PROGRAM Events
VAR
	Send_Start_Event : Send_Event_FB;
	Start_Event  : TcEventEntry := TC_Events.Pelletizer_Events.Start_Button_Event;
	
	Send_Stop_Event : Send_Event_FB;
	Stop_Event  : TcEventEntry := TC_Events.Pelletizer_Events.Stop_Button_Event;
//////////////////////////////////////////////////////////////////////////////////////////////////////////////////
	Send_EmergencyStop_Event : Send_Event_FB;
	EmergencyStop_Event : TcEventEntry := TC_Events.Pelletizer_Events.Emergency_Stop_Set_Event;

	Send_EmergencyStop_Reset_Event : Send_Event_FB;
	EmergencyStop_Reset_Event : TcEventEntry := TC_Events.Pelletizer_Events.Emergency_Stop_Reset_Event;
//////////////////////////////////////////////////////////////////////////////////////////////////////////////////
	Send_Discharge_Chute_NotPresent_Event : Send_Event_FB;
	Discharge_Chute_NotPresent_Event : TcEventEntry := TC_Events.Pelletizer_Events.Discharge_Chute_NotPresent_Event;
	
	Send_Discharge_Chute_Present_Event : Send_Event_FB;
	Discharge_Chute_Present_Event : TcEventEntry := TC_Events.Pelletizer_Events.Discharge_Chute_Present_Event;
//////////////////////////////////////////////////////////////////////////////////////////////////////////////////	
	Send_FeedThroat_NotPresent_Event : Send_Event_FB;
	FeedThroat_NotPresent_Event : TcEventEntry := TC_Events.Pelletizer_Events.FeedThroat_NotPresent_Event;
	
	Send_FeedThroat_Present_Event : Send_Event_FB;
	FeedThroat_Present_Event : TcEventEntry := TC_Events.Pelletizer_Events.FeedThroat_Present_Event;
//////////////////////////////////////////////////////////////////////////////////////////////////////////////////	
	Send_Feedroll_Drive_Fault_Event : Send_Event_FB;
	Feedroll_Drive_Fault_Event : TcEventEntry := TC_Events.Pelletizer_Events.Feedroll_Drive_Fault_Event;
	
	Send_Feedroll_Drive_Fault_Reset_Event : Send_Event_FB;
	Feedroll_Drive_Fault_Reset_Event : TcEventEntry := TC_Events.Pelletizer_Events.Feedroll_Drive_Fault_Reset_Event;
//////////////////////////////////////////////////////////////////////////////////////////////////////////////////	
	Send_Rotor_Drive_Fault_Event : Send_Event_FB;
	Rotor_Drive_Fault_Event : TcEventEntry := TC_Events.Pelletizer_Events.Rotor_Drive_Fault_Event;
	
	Send_Rotor_Drive_Fault_Reset_Event : Send_Event_FB;
	Rotor_Drive_Fault_Reset_Event : TcEventEntry := TC_Events.Pelletizer_Events.Rotor_Drive_Fault_Reset_Event;
//////////////////////////////////////////////////////////////////////////////////////////////////////////////////
	Send_Machine_Shutdown_Event : Send_Event_FB;
	Machine_Shutdown_Event : TcEventEntry := TC_Events.Pelletizer_Events.Machine_Shutdown_Event;	
	
	Send_Machine_PowerOn_Event : Send_Event_FB;
	Machine_PowerOn_Event : TcEventEntry := TC_Events.Pelletizer_Events.Machine_PowerOn_Event;
	First_Scan : BOOL := False;	
END_VAR

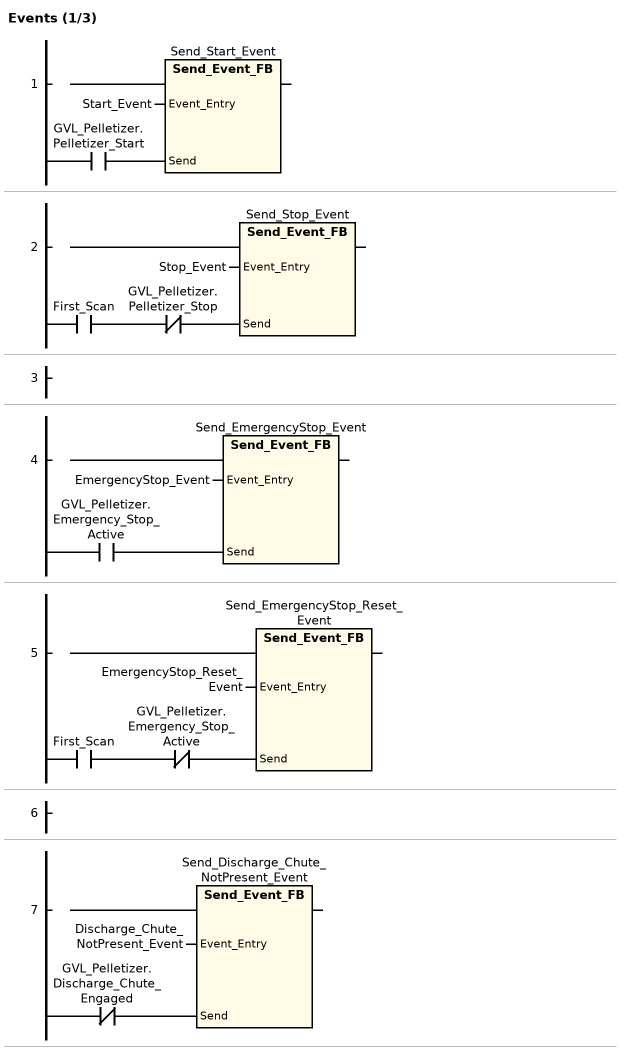
// NETWORK 1
Send_Start_Event(Event_Entry := Start_Event, Send := GVL_Pelletizer.Pelletizer_Start); // Send_Event_FB

// NETWORK 2
Send_Stop_Event(Event_Entry := Stop_Event, Send := First_Scan AND NOT GVL_Pelletizer.Pelletizer_Stop); // Send_Event_FB

// NETWORK 3

// NETWORK 4
Send_EmergencyStop_Event(Event_Entry := EmergencyStop_Event, Send := GVL_Pelletizer.Emergency_Stop_Active); // Send_Event_FB

// NETWORK 5
Send_EmergencyStop_Reset_Event(Event_Entry := EmergencyStop_Reset_Event, Send := First_Scan AND NOT GVL_Pelletizer.Emergency_Stop_Active); // Send_Event_FB

// NETWORK 6

// NETWORK 7
Send_Discharge_Chute_NotPresent_Event(Event_Entry := Discharge_Chute_NotPresent_Event, Send := NOT GVL_Pelletizer.Discharge_Chute_Engaged); // Send_Event_FB

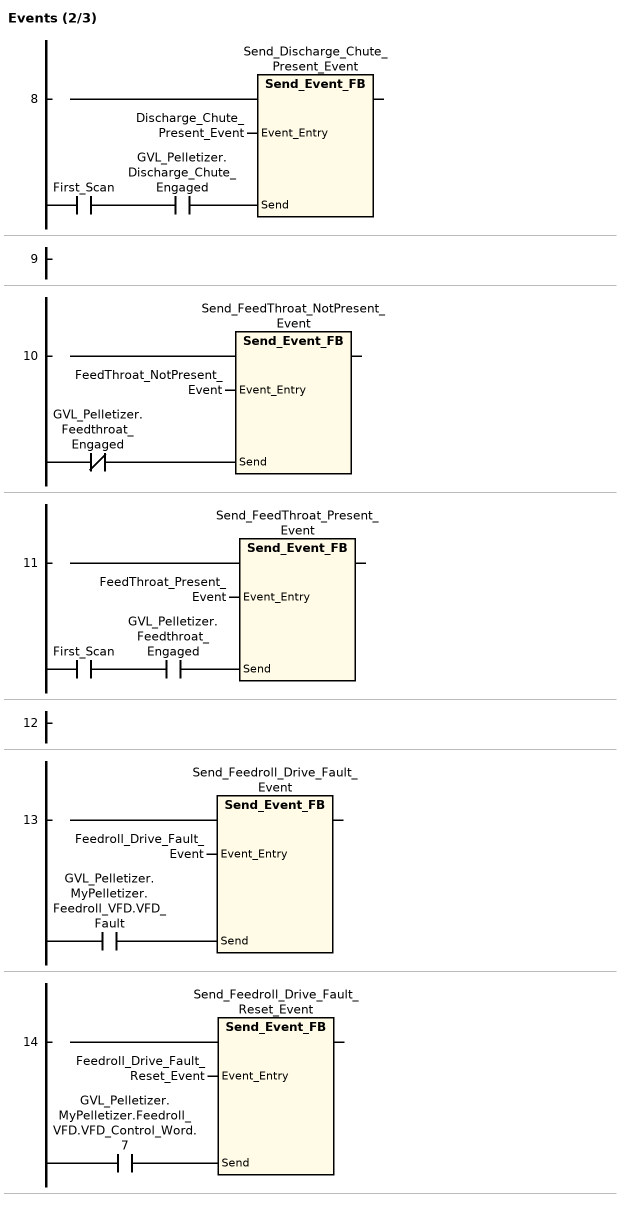
// NETWORK 8
Send_Discharge_Chute_Present_Event(Event_Entry := Discharge_Chute_Present_Event, Send := First_Scan AND GVL_Pelletizer.Discharge_Chute_Engaged); // Send_Event_FB

// NETWORK 9

// NETWORK 10
Send_FeedThroat_NotPresent_Event(Event_Entry := FeedThroat_NotPresent_Event, Send := NOT GVL_Pelletizer.Feedthroat_Engaged); // Send_Event_FB

// NETWORK 11
Send_FeedThroat_Present_Event(Event_Entry := FeedThroat_Present_Event, Send := First_Scan AND GVL_Pelletizer.Feedthroat_Engaged); // Send_Event_FB

// NETWORK 12

// NETWORK 13
Send_Feedroll_Drive_Fault_Event(Event_Entry := Feedroll_Drive_Fault_Event, Send := GVL_Pelletizer.MyPelletizer.Feedroll_VFD.VFD_Fault); // Send_Event_FB

// NETWORK 14
Send_Feedroll_Drive_Fault_Reset_Event(Event_Entry := Feedroll_Drive_Fault_Reset_Event, Send := GVL_Pelletizer.MyPelletizer.Feedroll_VFD.VFD_Control_Word.7); // Send_Event_FB

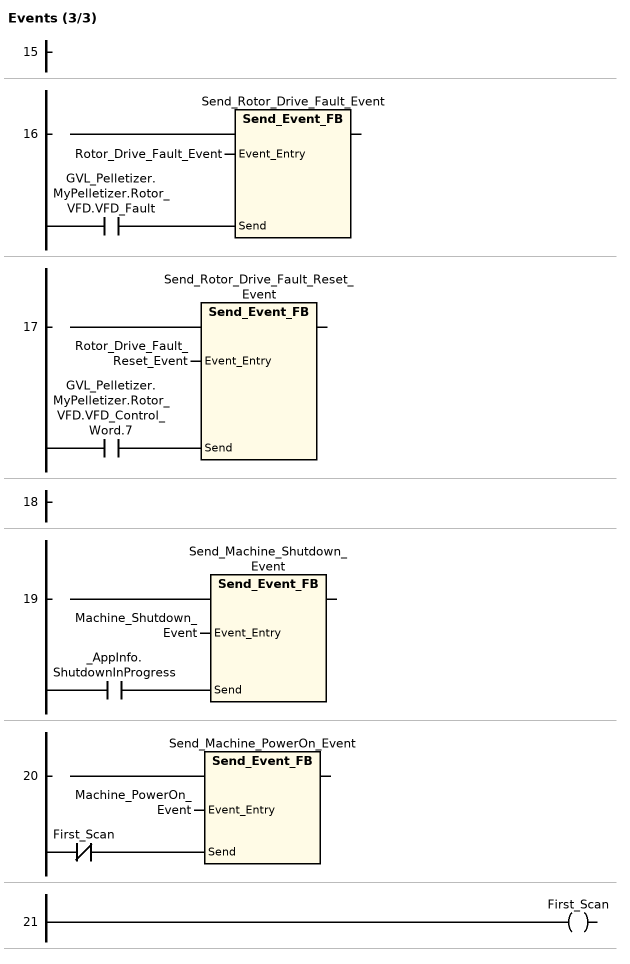
// NETWORK 15

// NETWORK 16
Send_Rotor_Drive_Fault_Event(Event_Entry := Rotor_Drive_Fault_Event, Send := GVL_Pelletizer.MyPelletizer.Rotor_VFD.VFD_Fault); // Send_Event_FB

// NETWORK 17
Send_Rotor_Drive_Fault_Reset_Event(Event_Entry := Rotor_Drive_Fault_Reset_Event, Send := GVL_Pelletizer.MyPelletizer.Rotor_VFD.VFD_Control_Word.7); // Send_Event_FB

// NETWORK 18

// NETWORK 19
Send_Machine_Shutdown_Event(Event_Entry := Machine_Shutdown_Event, Send := _AppInfo.ShutdownInProgress); // Send_Event_FB

// NETWORK 20
Send_Machine_PowerOn_Event(Event_Entry := Machine_PowerOn_Event, Send := NOT First_Scan); // Send_Event_FB

// NETWORK 21
First_Scan := TRUE;

END_PROGRAM

(* stored: Version 1.1.0.1, ProductVersion 3.1.4024.12
   POU Events: Id {bf716019-7947-4d54-948b-ddf8d1322a0f}, SpecialFunc None *)
